// TIA Portal V19 export
DATA_BLOCK "GlobalDB"   // DB9
{ S7_Optimized_Access := 'FALSE' }
   VAR RETAIN
      RTInfo : Struct   // Used to collect runtime information on an individual FB/FC
         Mode : UInt := 1;
         OBnumber : OB_ANY := 1;
         Info_LTIME : LTime := LT#0NS;
         RetVal : Int := 0;
      END_STRUCT;
      Runtime : Struct   // Used to collect individual runtime information of OB
         OB1Scan : Struct
            Min : LReal := 1000.0;
            Max : LReal;
            Current { ExternalAccessible := 'False'; ExternalVisible := 'False'; ExternalWritable := 'False'} : LReal;
            temp { ExternalAccessible := 'False'; ExternalVisible := 'False'; ExternalWritable := 'False'} : LReal;
            Mem { ExternalAccessible := 'False'; ExternalVisible := 'False'; ExternalWritable := 'False'} : LReal := 0.0;
            PreviousScan { ExternalAccessible := 'False'; ExternalVisible := 'False'; ExternalWritable := 'False'} : LReal;
            ResetMin : Bool;
            "Reset Max" : Bool;
         END_STRUCT;
      END_STRUCT;
      Trigger_StopSynch : Struct   // Used to trigger the Swapping of Status on the Reundant PLC
         REQ_FullSwapSequence { S7_SetPoint := 'True'} : Bool;   // Trigger used to perform a full swap of PLCs
         REQ_StopPrimary { S7_SetPoint := 'True'} : Bool;   // trigger a primary stop
         REQ_SynchUp { S7_SetPoint := 'True'} : Bool;   // trigger a synchronization
         Mode_StopPrimary : Int := 8;   // Stop Primary = 8
         Mode_SynchUp : Int := 7;   // Synchronization = 7
         StopPrimary_Retry_Busy : Bool;   // triggered due to RHCTRL being busy
         SynchUp_Retry_Busy : Bool;   // triggered due to RHCTRL being busy
         SyncSequenceFlag : Bool;
         RH_CTRL_PrimaryStop : Struct   // Used to stop and synch primary or backup
            REQ : Bool;
            Ret_Val : Byte;
            Busy : Bool;
         END_STRUCT;
         RH_CTRL_SyncUp : Struct   // Used to stop and synch primary or backup
            REQ : Bool;
            Ret_Val : Byte;
            Busy : Bool;
         END_STRUCT;
         SyncSequenceTimer : IEC_TIMER;
         SequenceTimer : IEC_TIMER;   // Timer to sequence between stop and synch
         SequenceAlarm { S7_SetPoint := 'True'} : Bool;
      END_STRUCT;
      Network { S7_SetPoint := 'True'} : "NetworkSwitchHMI";   // Used to collect switch XC208 details
      SystemTime { S7_SetPoint := 'True'} : DTL;   // Used to record cycle time of code
      tempSystemTime { S7_SetPoint := 'True'} : Int;
      "Array" : Array[0..1000] of "typeDiagnostics";   // Test Array
   END_VAR
BEGIN
   Trigger_StopSynch.SequenceTimer.PT := T#25s;   // Time based on full sequence elapsed timer
END_DATA_BLOCK
